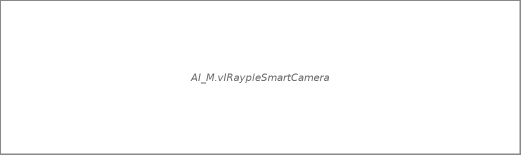
VISUALIZATION vWeighingTunelVisionFrame  // 521x155
    Frame (0,0 521x155)
        shows AI_M.vIRaypleSmartCamera(fb := MAIN.fbSmartCamera)
END_VISUALIZATION

(* stored: Version 1.1.0.1, ProductVersion 3.1.4024.16
   Visu vWeighingTunelVisionFrame: Id {6b7092fc-17c1-46aa-8e26-504e88321950} *)
